Staubli VAL3: CheckAxis.pgx

public program CheckAxis(bool& x_b7Axis, bool& x_b8Axis)
begin

 x_b7Axis=$XgetNbAxes()>=1
 x_b8Axis=$XgetNbAxes()>=2


end
